TYPE (* IEC61131-3, Table 14#5 *)
  (* Standard: 1131-3 *)
  (* Version 0.0, 1/8/2024, Cheyan, Schneider Electric, Template *)
  PACKAGE Main;
  {SET_ATTRIBUTE(nxtDataType, z/yCPi5cyPDsYuYBrz+XyN166j18T5K4J2Q3xaJpnrNfQWJwFVk0wNWrZu5DnBj5bF0C1aNk6OB1CUwVj8gW42LZr/I8KdMo17tDavdvsGG6DhN/811gPwZegzo+YN9HUJM+RBxfMAI=)}
  INS : STRUCT
    stVal : DINT;
    q : Quality;
    t : TimeStamp;
  END_STRUCT;
END_TYPE
